(* PLC project static_torsion.project, CODESYS CODESYS V3.5 SP17 Patch 3 *)
(* stored: creationDateTime 1970-01-01T00:00:00, modificationDateTime 2026-06-22T15:12:39.4699931 *)

FUNCTION GetCommand : WORD
  VAR_INPUT
    control_word : S_CTRL;
  END_VAR
  VAR
    out : WORD;
  END_VAR

            out.0 := control_word.cmd_bit0;
out.1 := control_word.cmd_bit1;
out.2 := control_word.cmd_bit2;

GetCommand := out;


          
END_FUNCTION
